PROGRAM SchedulerPublicHolidays
VAR
	fbHVACSchedulerPublicHolidays:FB_HVACSchedulerPublicHolidays;
	eDataSecurityType:E_HVACDataSecurityType;
	bSetDefault:BOOL;
	bEnable:BOOL;
	dtSystemTime:DT;
	bReset:BOOL;
	arrHoliday:ARRAY[1..20] OF ST_HVACHoliday;
	bOutput:BOOL;
	bEdgeOn:BOOL;
	bEdgeOff:BOOL;
	tNextOn:TIME;
	tNextOff:TIME;
	bInvalidParameter:BOOL;
END_VAR

fbHVACSchedulerPublicHolidays(
	eDataSecurityType:=eDataSecurityType , 
	bSetDefault:= bSetDefault, 
	bEnable:=bEnable, 
	dtSystemTime:=dtSystemTime, 
	bReset:=bReset, 
	arrHoliday:=arrHoliday, 
	bOutput=>bOutput, 
	bEdgeOn=>bEdgeOn, 
	bEdgeOff=>bEdgeOff, 
	tNextOn=>tNextOn, 
	tNextOff=>tNextOff, 
	bInvalidParameter=>bInvalidParameter);

END_PROGRAM

(* stored: Version 1.1.0.1, ProductVersion 3.1.4024.3
   POU SchedulerPublicHolidays: Id {fdb4eade-21d2-43fb-9056-12e64699a412}, SpecialFunc None *)
